{attribute 'qualified_only'}
{attribute 'strict'}
{attribute 'to_string'}
TYPE TASK_PROCESSING_RESULT :
(
	IN_PROGRESS := 0,
	DONE := 1,
	ABORTED := 2
);
END_TYPE

(* stored: Version 1.1.0.1
   DUT TASK_PROCESSING_RESULT: Id {a9122e0d-49af-4bce-9974-60ec7c2b7dcc} *)
